PROGRAM PRG_FactoryIO_ModbusTCP_Write
// Dépendance Tc2_ModbusSrv (TF6250-Modbus-TCP)
// FB_Bool_To_Word + FB_Word_To_Bool
VAR
	fb_FactoryIO_ModbusTCP : FB_FactoryIO_ModbusTCP;
END_VAR

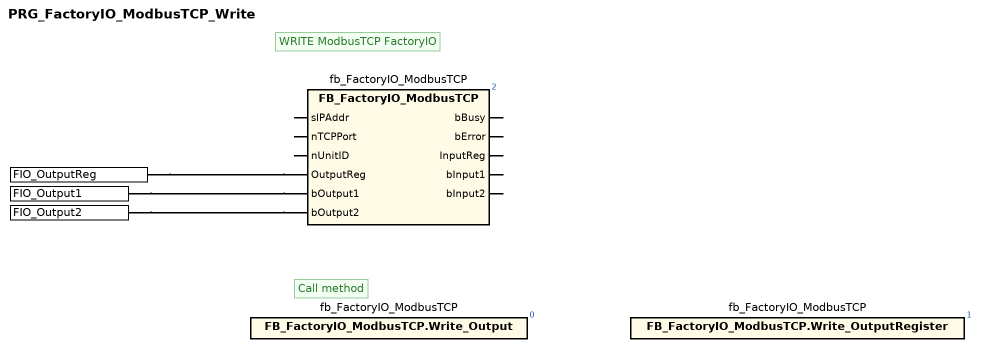
// Call method
fb_FactoryIO_ModbusTCP.Write_Output();
fb_FactoryIO_ModbusTCP.Write_OutputRegister();
// WRITE ModbusTCP FactoryIO
fb_FactoryIO_ModbusTCP(OutputReg := FIO_OutputReg, bOutput1 := FIO_Output1, bOutput2 := FIO_Output2);

END_PROGRAM

(* stored: Version 1.1.0.1, ProductVersion 3.1.4024.11
   POU PRG_FactoryIO_ModbusTCP_Write: Id {86f813b4-6ada-4788-8afc-fe1c48f3163b}, SpecialFunc None *)
